# B&R Automation Studio project lab_1
Automation Studio 4.5.2.102

## Configuration Config1

CPU 4PP065.0571-P74, AutomationRuntime D4.52, Build 4.1.2, Vc V4.52.0, Safety 1.10

### Task classes (Cpu.sw)
```
Cyclic#1:
  Program <- Program.prg
Binaries: udbdef, TCData, arsvcreg, iomap, ashwac, Role, sysconf, arconfig, asfw, ashwd, User
Libraries: McBase, Library
```

### Hardware
```
4PP065_0571_P74 : 4PP065.0571-P74 v1.1.2.0
  Connector IF5:
    ActivateDevice = 1
    Mode = Manual
    InternetAddress = 127.0.0.1
    SubnetMask = 255.255.255.0
  ConfigurationID = labBR
  Simulation = 1
```

## Logical view

Binary libraries used (declarations not repeated): operator, runtime, astime, AsIecCon, McBase

### Library Logical/Libraries/Library (ANSIC)

#### Library.fun - Exported functions and function blocks
```iecst
{REDUND_ERROR} FUNCTION_BLOCK FB_integrator (*TODO: Add your comment here*) (*$GROUP=User,$CAT=User,$GROUPICON=User.png,$CATICON=User.png*)
	VAR_INPUT
		in : {REDUND_UNREPLICABLE} REAL;
		dt : REAL;
	END_VAR
	VAR
		prev_value : REAL;
	END_VAR
	VAR_OUTPUT
		out : {REDUND_UNREPLICABLE} REAL;
	END_VAR
END_FUNCTION_BLOCK

{REDUND_ERROR} FUNCTION_BLOCK FB_Motor (*TODO: Add your comment here*) (*$GROUP=User,$CAT=User,$GROUPICON=User.png,$CATICON=User.png*)
	VAR_INPUT
		u : {REDUND_UNREPLICABLE} REAL;
		dt : REAL;
	END_VAR
	VAR
		ke : {REDUND_UNREPLICABLE} REAL;
		Tm : {REDUND_UNREPLICABLE} REAL;
		integrator : {REDUND_UNREPLICABLE} FB_integrator;
	END_VAR
	VAR_OUTPUT
		w : {REDUND_UNREPLICABLE} REAL;
		phi : {REDUND_UNREPLICABLE} REAL;
	END_VAR
END_FUNCTION_BLOCK

{REDUND_ERROR} FUNCTION_BLOCK FB_Controler (*TODO: Add your comment here*) (*$GROUP=User,$CAT=User,$GROUPICON=User.png,$CATICON=User.png*)
	VAR_INPUT
		e_in : {REDUND_UNREPLICABLE} REAL;
		dt : REAL;
	END_VAR
	VAR
		sum : {REDUND_UNREPLICABLE} REAL;
		integrator : {REDUND_UNREPLICABLE} FB_integrator;
		k_p : {REDUND_UNREPLICABLE} REAL;
		k_i : {REDUND_UNREPLICABLE} REAL;
		max_abs_value : {REDUND_UNREPLICABLE} REAL;
		iyOld : {REDUND_UNREPLICABLE} REAL;
		a : {REDUND_UNREPLICABLE} REAL;
		e_kp : {REDUND_UNREPLICABLE} REAL;
	END_VAR
	VAR_OUTPUT
		u : {REDUND_UNREPLICABLE} REAL;
	END_VAR
END_FUNCTION_BLOCK
```

#### FB_Integrator.c
```c
#include <bur/plctypes.h>
#ifdef __cplusplus
	extern "C"
	{
#endif
	#include "Library.h"
#ifdef __cplusplus
	};
#endif
/* TODO: Add your comment here */
void FB_integrator(struct FB_integrator* inst)
{
	/*TODO: Add your code here*/
	inst->dt = d_t;
	inst->out = inst->dt * inst->in + inst->prev_value;
	inst->prev_value = inst->out;
}
```

#### FB_Motor.c
```c
#include <bur/plctypes.h>
#ifdef __cplusplus
	extern "C"
	{
#endif
	#include "Library.h"
#ifdef __cplusplus
	};
#endif
/* TODO: Add your comment here */
void FB_Motor(struct FB_Motor* inst)
{
	REAL a = (inst->u / inst->ke) - inst->w;
	REAL b = a / inst->Tm;

	inst->integrator.in = b;
	FB_integrator(&inst->integrator);

	inst->w = inst->integrator.out;

	inst->integrator.in = inst->w;
	FB_integrator(&inst->integrator);

	inst->phi = inst->integrator.out;
}
```

#### FB_Controler.c
```c
#include <bur/plctypes.h>
#ifdef __cplusplus
	extern "C"
	{
#endif
	#include "Library.h"
#ifdef __cplusplus
	};
#endif
/* TODO: Add your comment here */
void FB_Controler(struct FB_Controler* inst)
{
	/*TODO: Add your code here*/
	REAL a = inst->e_in * inst->k_p;
	REAL b = inst->e_in * inst->k_i;

	//ограничение напряжения
	a = a > inst->max_abs_value ?  inst->max_abs_value : a;
	a = a < -inst->max_abs_value ? -inst->max_abs_value : a;

	inst->integrator.in = b + inst->sum;
	FB_integrator(&inst->integrator);

	REAL sum = a + inst->integrator.out;
	inst->u = sum;

	inst->u = sum;

	inst->u = inst->u > inst->max_abs_value ? inst->max_abs_value : inst->u;
	inst->u = inst->u < -inst->max_abs_value ? -inst->max_abs_value : inst->u;

	inst->sum = inst->u - sum;

//	if(abs(a) < inst->max_abs_value)
//	{
//		a = a;
//	}
//	else
//	{
//		if(a < 0)
//		{
//			a = (-1)*inst->max_abs_value
//		}
//		else
//		{
//			a = inst->max_abs_value
//		}
//	}
}
```

### Program Logical/Program

#### Variables.var
```iecst
VAR
	fb_controller : FB_Controler;
	fb_motor1 : FB_Motor;
	fb_motor2 : FB_Motor;
	speed : REAL;
	counter : UINT;
	enable : BOOL;
END_VAR
```

#### Main.c
```c
#include <bur/plctypes.h>

#ifdef _DEFAULT_INCLUDES
	#include <AsDefault.h>
#endif

void _INIT ProgramInit(void)
{
	fb_motor1.ke = 0.24;//1.18; //0.24
	fb_motor1.Tm = 0.1;//0.17;//0.1
	fb_motor1.u = 0;
	fb_motor1.dt = 0.01;

	fb_motor2.ke = 0.24;
	fb_motor2.Tm = 0.1;
	fb_motor2.u = 0;
	fb_motor2.dt = 0.01;

	fb_controller.k_p = 0.78;
	fb_controller.k_i = 7.2;
	fb_controller.max_abs_value = 24.0;
	fb_controller.dt = 0.01;

	speed = 0;
	counter = 0;
	enable = 0;
}

void _CYCLIC ProgramCyclic(void)
{
	if(enable)
	{
		if(counter == 200)
		{
			speed = 0;
			counter = 0;
		}
		else if(counter == 50)
		{
			speed = 50;
		}
		fb_controller.e_in = speed - fb_motor1.w;
		FB_Controler(&fb_controller);

		fb_motor1.u = fb_controller.u;
		FB_Motor(&fb_motor1);

		fb_motor2.u = speed * fb_motor2.ke;
		FB_Motor(&fb_motor2);

		counter++;
	}
}

void _EXIT ProgramExit(void)
{

}
```

Listed in the project but not available here: Logical/Libraries/Library/Types.typ, Logical/Libraries/Library/Constants.var
